{attribute 'GeneratedUsingTerminal: EL4024-0000-0018'}
{attribute addProperty BoxType "EL4024-0000-0018"}
{attribute addProperty Id "EtcSlaveTerminalBaseAO_Output_Channel_1AT %Q*AO_Output_Channel_BA7EBB7C2AO_Output_Channel_2AT %Q*AO_Output_Channel_BA7EBB7C2AO_Output_Channel_3AT %Q*AO_Output_Channel_BA7EBB7C2AO_Output_Channel_4AT %Q*AO_Output_Channel_BA7EBB7C2WcStateAT %I*WcState_0B2B16F91InfoDataAT %I*InfoData_32EB74EA10"}
{attribute addProperty CRC "3361817969"}
{attribute addProperty Size "19"}
TYPE EL4024_C8614571 EXTENDS EtcSlaveTerminalBase :
STRUCT
	{attribute addProperty Name "AO_Output_Channel_1"}
	AO_Output_Channel_1 : AO_Output_Channel_BA7EBB7C;
	{attribute addProperty Name "AO_Output_Channel_2"}
	AO_Output_Channel_2 : AO_Output_Channel_BA7EBB7C;
	{attribute addProperty Name "AO_Output_Channel_3"}
	AO_Output_Channel_3 : AO_Output_Channel_BA7EBB7C;
	{attribute addProperty Name "AO_Output_Channel_4"}
	AO_Output_Channel_4 : AO_Output_Channel_BA7EBB7C;
	{attribute addProperty Name "WcState"}
	WcState : WcState_0B2B16F9;
	{attribute addProperty Name "InfoData"}
	InfoData : InfoData_32EB74EA;
END_STRUCT
END_TYPE

(* stored: Version 1.2.0.0, ProductVersion 3.1.4024.9
   DUT EL4024_C8614571: Id {112bcc58-124a-4037-99a6-bd3980a1b783} *)
